(* CoDeSys 2.3.9.37 project: Cap7_1.pro *)
(* Libraries: Standard.LIB 4.10.05 12:14:46 *)

(* Global variable list: Global_Variables *)
VAR_GLOBAL

(* Variables de entrada *)
	N1:BOOL;
      N2:BOOL;
      DS:BOOL;
      DI:BOOL;
(* Variables de salida *)
 	Bomba1:BOOL;
  	Bomba2:BOOL;

END_VAR

(* POU PLC_PRG, IL *)
PROGRAM PLC_PRG
VAR
END_VAR

END_PROGRAM

(* Visualisation Combi1
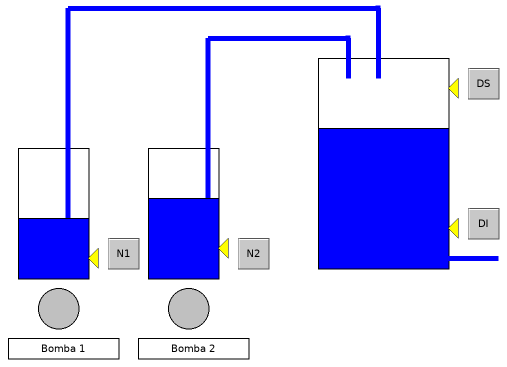
ellipse at (100,320)-(141,361): alarm colour if Bomba1
button at (170,270)-(201,301): text "N1"; toggles N1
button at (300,270)-(331,301): text "N2"; toggles N2
button at (530,100)-(561,131): text "DS"; toggles DS
button at (530,240)-(561,271): text "DI"; toggles DI
rectangle at (70,370)-(181,391): text "Bomba 1"
ellipse at (230,320)-(271,361): alarm colour if Bomba2
rectangle at (200,370)-(311,391): text "Bomba 2"
15 more shapes without text or variables
*)
